(* PLC project bottle, Dassault Systèmes ControlBuild 2024x Refresh1 *)
(* stored: creationDateTime 2024-01-24T08:52:15-01:00 *)

CONFIGURATION bottle
  VAR_GLOBAL
    simuperiod : REAL := 50000.0;
    taskname : STRING(50) := 'bottle.exe';
    allowpreconditions : BOOL := true;
    allowpostconditions : BOOL := true;
  END_VAR
END_CONFIGURATION
